{attribute 'no_explicit_call' := 'Do not call the body - Stick to OOP'}
FUNCTION_BLOCK FB_XTS_Mover EXTENDS FB_CH_Object IMPLEMENTS I_XTS_Mover, I_XTS_Mover_PLC
VAR	
	//Link to NC
	Axis : FB_XTS_Axis;

	{attribute 'hide'}
	bInitDone : BOOL;
	{attribute 'hide'}
	ipXtsSystem : I_XTS_System_Registration;
	{attribute 'hide'}
	ipUtilityMover : I_TcIoXtsXpuMover;
	{attribute 'hide'}
	ipProductData : I_XTS_ProductData; //later the required interface of the tool or product can be queried via query interface
	{attribute 'hide'}
	ipParentStation : I_XTS_Station; //This is the station in which the Mover is currently standing or moving.	
	{attribute 'hide'}
	ipNextMover : I_XTS_Mover;
	{attribute 'hide'}
	sTargedStation : STRING;
	{attribute 'hide'}
	fLastCmdTargedPosition : LREAL; //the last commanded target position [mm]
	{attribute 'hide'}
	fLastCmdTargedVelocity : LREAL; //the last commanded target speed
	{attribute 'hide'}	
	fLastCmdTargedGap 	: LREAL; //the last commanded target gap
	{attribute 'hide'}
	bInGroup : BOOL;	
	{attribute 'hide'}	
	lrTrackLentgh 			: LREAL; //[mm]  Modulo
	{attribute 'hide'}
	fbFeedback 					: CHALET_BaseComponents.FB_CH_Feedback(ipSourceInfo := fbSourceInfo);;
	
END_VAR
VAR PERSISTENT
	fDrivenDistance : LREAL;
END_VAR

{attribute 'monitoring':='call'}
PROPERTY Coupled : BOOL
GET
Coupled := THIS^.Axis.Coupled;
END_GET
END_PROPERTY

{attribute 'OPC.UA.DA.Property' := '1'}
{attribute 'monitoring':='call'}
PROPERTY DefaultAcceleration : LREAL
GET
DefaultAcceleration := THIS^.Axis.DefaultAcceleration;
END_GET
SET
THIS^.Axis.DefaultAcceleration := DefaultAcceleration;
END_SET
END_PROPERTY

{attribute 'OPC.UA.DA.Property' := '1'}
{attribute 'monitoring':='call'}
PROPERTY DefaultDeceleration : LREAL
GET
DefaultDeceleration := THIS^.Axis.DefaultDeceleration;
END_GET
SET
THIS^.Axis.DefaultDeceleration := DefaultDeceleration;
END_SET
END_PROPERTY

{attribute 'OPC.UA.DA.Property' := '1'}
{attribute 'monitoring':='call'}
PROPERTY DefaultJerk : LREAL
GET
DefaultJerk := THIS^.Axis.DefaultJerk;
END_GET
SET
THIS^.Axis.DefaultJerk := DefaultJerk;
END_SET
END_PROPERTY

METHOD Disable : HRESULT
Axis.PowerOff();


//Show as feedback the state of the includet axis
fbFeedback.ActiveCommand := Axis.Feedback.ActiveCommand;
fbFeedback.LastCommandAccepted := Axis.Feedback.LastCommandAccepted;
fbFeedback.HR := Axis.Feedback.hr;


IF Axis.Feedback.LastCommandAccepted THEN
	Disable := S_OK;
ELSE  
	Disable := E_FAIL;;	
END_IF
END_METHOD

{attribute 'monitoring':='call'}
PROPERTY DrivenDistance : LREAL
GET
DrivenDistance := fDrivenDistance;
END_GET
END_PROPERTY

METHOD Enable : HRESULT
Axis.PowerOn();


//Show as feedback the state of the includet axis
fbFeedback.ActiveCommand := Axis.Feedback.ActiveCommand;
fbFeedback.LastCommandAccepted := Axis.Feedback.LastCommandAccepted;
fbFeedback.HR := Axis.Feedback.hr;


IF Axis.Feedback.LastCommandAccepted THEN
	Enable := S_OK;
ELSE  
	Enable := E_FAIL;;	
END_IF
END_METHOD

METHOD FB_init : BOOL
VAR_INPUT
	bInitRetains : BOOL; // if TRUE, the retain variables are initialized (warm start / cold start)
	bInCopyCode : BOOL;  // if TRUE, the instance afterwards gets moved into the copy code (online change)
	
	ipXtsSystem : I_XTS_System_Registration; //Interface to XTS system object
END_VAR
VAR_INST
	{attribute 'hide'}
	bFBInitCalledOnce : BOOL; //Do the following code once during start up and not during onlinechange
END_VAR
//Do the following code once during start up and not during onlinechange
IF NOT bFBInitCalledOnce THEN 
	

	//Regristrate object in System
	IF ipXtsSystem <> 0 THEN
		ipXtsSystem.RegisterMover(THIS^);
		THIS^.ipXtsSystem := ipXtsSystem;
	END_IF


	
END_IF

bFBInitCalledOnce := TRUE;
END_METHOD

{attribute 'monitoring':='call'}
PROPERTY Feedback : I_CH_Feedback
GET
Feedback := THIS^.fbFeedback;
END_GET
END_PROPERTY

(*The _ PLC interface provides the user with a simplified interface for commanding between the stations. Sometimes, however, this is not enough. 
Either you get the corresponding interface with the __Queryinterface or you can get full access with this property.*)
PROPERTY FullAccess : I_XTS_Mover
GET
FullAccess := (THIS^);
END_GET
END_PROPERTY

PROPERTY getAxisRef : REFERENCE TO Tc2_MC2.AXIS_REF
GET
getAxisRef REF= THIS^.Axis.getAxisRef;
END_GET
END_PROPERTY

METHOD HaltCA : HRESULT
VAR_INPUT
END_VAR
Axis.HaltCA(
	fDeceleration:= 0, //use default
	fJerk:= 0, //use default
	fGap:= fLastCmdTargedGap);
	

//Show as feedback the state of the includet axis
fbFeedback.ActiveCommand := Axis.Feedback.ActiveCommand;
fbFeedback.LastCommandAccepted := Axis.Feedback.LastCommandAccepted;
fbFeedback.HR := Axis.Feedback.hr;


IF Axis.Feedback.LastCommandAccepted THEN
	HaltCA := S_OK;
ELSE  
	HaltCA := E_FAIL;;	
END_IF
END_METHOD

PROPERTY IdentInGroup : IDENT_IN_GROUP_REF
GET
IdentInGroup := UDINT_TO_IDENTINGROUP(THIS^.Axis.getAxisRef.NcToPlc.AxisId);
END_GET
END_PROPERTY

METHOD Initialize : HRESULT
VAR

END_VAR
fbFeedback.hr := S_OK;	

IF NOT THIS^.bInitDone THEN
	fbFeedback.ActiveCommand := 'Init';
	
	//Get Tracklength from system
	THIS^.lrTrackLentgh := THIS^.ipXtsSystem.TrackLength;
	
	
	//Validate Settings
	IF (lrTrackLentgh <= 0) THEN
		fbFeedback.hr := GetMostSignificant(fbFeedback.hr, E_FAIL);		
	END_IF
	

	//If only one mover is in project, then interface stays 0.
	IF THIS^.ipXtsSystem.Movers.Size > 1 THEN
		THIS^.ipNextMover := THIS^.ipXtsSystem.getMoverInFront(THIS^);
		//Validate Settings
		IF (ipNextMover = 0) THEN
			fbFeedback.hr := GetMostSignificant(fbFeedback.hr, E_FAIL);	
		END_IF
	ELSE
		THIS^.ipNextMover := 0;
	END_IF
	
	// Get XTS Utility mover object
	IF ipXtsSystem.Environment <> 0 THEN
		ipUtilityMover := ipXtsSystem.Environment.UtilityEnvirement.GetMoverInterfaceByAxisId(THIS^.getAxisRef.NcToPlc.AxisId);
		//Validate 
		IF (ipUtilityMover = 0) THEN
			fbFeedback.hr := GetMostSignificant(fbFeedback.hr, E_FAIL);	
		END_IF
	END_IF
	
	
	//InitAxis
	fbFeedback.hr := GetMostSignificant(fbFeedback.hr, Axis.Initialize());	

	bInitDone := CheckOk(fbFeedback.hr);
END_IF

Initialize := fbFeedback.hr;
END_METHOD

{attribute 'monitoring':='call'}
PROPERTY LagDistance : LREAL
GET
LagDistance := THIS^.Axis.LagDistance;
END_GET
END_PROPERTY

{attribute 'monitoring':='call'}
PROPERTY LastCmdTargedGap : LREAL
GET
LastCmdTargedGap := fLastCmdTargedGap;
END_GET
END_PROPERTY

{attribute 'monitoring':='call'}
PROPERTY LastCmdTargedPosition : LREAL
GET
LastCmdTargedPosition := fLastCmdTargedPosition;
END_GET
END_PROPERTY

{attribute 'monitoring':='call'}
PROPERTY LastCmdTargedVelocity : LREAL
GET
LastCmdTargedVelocity := fLastCmdTargedVelocity;
END_GET
END_PROPERTY

METHOD MoveAbsCA : HRESULT
VAR_INPUT
	fPosition	: LREAL := MC_INVALID;
	fVelocity	: LREAL := MC_INVALID;
	fGap		: LREAL := MC_DEFAULT;
	eDirection	: Tc3_Mc3Definitions.MC_DIRECTION;
END_VAR
Axis.MoveAbsoluteCA(
	fPosition:= fPosition, 
	fVelocity:= fVelocity, 
	fGap:= fGap, 
	fAcceleration:= 0, //Use Axis default
	fDeceleration:= 0, //Use Axis default
	fJerk:= 0, 			//Use Axis default
	eDirection := eDirection,
	eBufferMode:= Tc3_Mc3Definitions.MC_BUFFER_MODE.mcAborting);

THIS^.fLastCmdTargedVelocity := fVelocity;
THIS^.fLastCmdTargedPosition := fPosition;
THIS^.fLastCmdTargedGap := fGap;


//Show as feedback the state of the includet axis
fbFeedback.ActiveCommand := Axis.Feedback.ActiveCommand;
fbFeedback.LastCommandAccepted := Axis.Feedback.LastCommandAccepted;
fbFeedback.HR := Axis.Feedback.hr;


IF Axis.Feedback.LastCommandAccepted THEN
	MoveAbsCA := S_OK;
ELSE  
	MoveAbsCA := E_FAIL;;	
END_IF
END_METHOD

{attribute 'monitoring':='call'}
PROPERTY MoverInGroup : BOOL
GET
MoverInGroup := bInGroup;
END_GET
SET
bInGroup := MoverInGroup;
END_SET
END_PROPERTY

{attribute 'monitoring':='call'}
PROPERTY Moving : BOOL
GET
Moving := THIS^.Axis.Moving;
END_GET
END_PROPERTY

{attribute 'monitoring':='call'}
PROPERTY NextMover : I_XTS_Mover
GET
NextMover := ipNextMover;
END_GET
END_PROPERTY

{attribute 'monitoring':='call'}
PROPERTY OID : OTCID
GET
OID := THIS^.Axis.OID;
END_GET
END_PROPERTY

{attribute 'monitoring':='call'}
PROPERTY ParentStation : I_XTS_Station
GET
ParentStation := ipParentStation;
END_GET
SET
ipParentStation := ParentStation;
END_SET
END_PROPERTY

{attribute 'monitoring':='call'}
PROPERTY PositionOnTrack : LREAL
GET
//Round to 3 digits. If Axis is not enabled, use act position
IF THIS^.Axis.getAxisRef.Status.Disabled THEN
	PositionOnTrack := TO_LREAL(TRUNC(THIS^.Axis.ActPosModulo*1000))/1000;
ELSE
	PositionOnTrack := TO_LREAL(TRUNC(THIS^.Axis.SetPosModulo*1000))/1000;	
END_IF
END_GET
END_PROPERTY

{attribute 'monitoring':='call'}
PROPERTY PUBLIC ProductData : I_XTS_ProductData
GET
ProductData := ipProductData;
END_GET
SET
// No change. Same interface is set again
IF ipProductData = ProductData THEN
	;//Noting
	
ELSE

	// If allready an interface is linked. Unlink
	IF ipProductData <> 0 THEN
		ipProductData.LinkToMover(0);
		ipProductData := 0;
	END_IF
	
	// Link and store new interface
	IF ProductData <> 0 THEN
		ProductData.LinkToMover(THIS^);
		ipProductData := ProductData;
	END_IF
END_IF
END_SET
END_PROPERTY

METHOD Reset : HRESULT
Axis.Reset();

//Show as feedback the state of the includet axis
fbFeedback.ActiveCommand := Axis.Feedback.ActiveCommand;
fbFeedback.LastCommandAccepted := Axis.Feedback.LastCommandAccepted;
fbFeedback.HR := Axis.Feedback.hr;


IF Axis.Feedback.LastCommandAccepted THEN
	Reset := S_OK;
ELSE  
	Reset := E_FAIL;;	
END_IF
END_METHOD

{attribute 'monitoring':='call'}
PROPERTY SetAcceleration : LREAL
GET
SetAcceleration := THIS^.Axis.SetAcceleration;
END_GET
END_PROPERTY

{attribute 'monitoring':='call'}
PROPERTY SetVelocity : LREAL
GET
SetVelocity := THIS^.Axis.SetVelocity;
END_GET
END_PROPERTY

{attribute 'monitoring':='call'}
PROPERTY TargedStation : STRING
GET
TargedStation := sTargedStation;
END_GET
SET
sTargedStation := TargedStation;
END_SET
END_PROPERTY

METHOD Update : HRESULT
VAR
	fDistanceThisCycle : LREAL;
END_VAR
VAR_INST
	fLastMoverPosition : LREAL;
END_VAR
// Total distance traveled by the mover
IF Axis.Moving THEN
	fDistanceThisCycle := ABS(Axis.SetPosModulo-fLastMoverPosition);
	IF fDistanceThisCycle > (THIS^.lrTrackLentgh*0.5) THEN
		fDistanceThisCycle := THIS^.lrTrackLentgh-fDistanceThisCycle;
	END_IF
	fDrivenDistance := fDrivenDistance + fDistanceThisCycle;
END_IF

fLastMoverPosition := Axis.SetPosModulo;

Axis.Update();

//Show as feedback the state of the includet axis
fbFeedback.ActiveCommand := Axis.Feedback.ActiveCommand;
fbFeedback.HR := Axis.Feedback.hr;
END_METHOD

{attribute 'monitoring':='call'}
PROPERTY UtilityMover : I_TcIoXtsXpuMover
GET
UtilityMover := ipUtilityMover;
END_GET
END_PROPERTY

END_FUNCTION_BLOCK

(* stored: Version 1.1.0.1, ProductVersion 3.1.4024.12
   POU FB_XTS_Mover: Id {3ed790a4-6e64-4b54-8db7-341624f96fe6}, SpecialFunc None
   Folder Command: Id {ca288374-806c-40ea-bc74-0ab5bbcbeeac}
   Folder Dynamics: Id {b9fcfb38-b272-4ca4-b13a-341f5f54d90d}
   Folder Status: Id {36fbca5a-40fa-4fee-a207-226360d4b0d4}
   Property Coupled: Id {627291ab-402b-4929-a093-0ff8fc3ea751}
   Get Get: Id {f28a9d3d-b665-4255-8ee8-a1611de68e13}
   Property DefaultAcceleration: Id {18610012-8a94-4ab6-bb6e-6d4fcc935be7}
   Get Get: Id {30c1feb4-1bec-4b32-8312-941a2f3f97e6}
   Set Set: Id {73641ac0-c47d-4373-aafd-c8aa42e11a4f}
   Property DefaultDeceleration: Id {a4e01ee3-7720-44ba-aa6b-afa8d7117cca}
   Get Get: Id {ff90a48b-809c-4768-9581-05a95fc76f54}
   Set Set: Id {ecb6ccf7-e313-4889-af0f-b2b90db416f6}
   Property DefaultJerk: Id {d2dd93df-7379-493e-a0e2-335666e5944c}
   Get Get: Id {9bcab0a6-60f8-42f0-9374-f84d6b198092}
   Set Set: Id {5eea3280-3211-4781-b593-3f1678c35bbf}
   Method Disable: Id {fabc84ce-66bc-42ad-9f05-26b65256e1b0}
   Property DrivenDistance: Id {b520ba11-eae3-4194-b965-36b18e5c7ced}
   Get Get: Id {713472d5-7bea-4713-b937-1508a3c15ef1}
   Method Enable: Id {c5208f99-fcd6-4588-ba54-a943e08cbd2d}
   Method FB_init: Id {26d010fc-cadf-4788-a716-5e39c9198509}
   Property Feedback: Id {78e76366-75b3-4e4d-b82e-9b66faf8cccb}
   Get Get: Id {53c4eaab-cafe-47f9-880a-ceebaeabf33e}
   Property FullAccess: Id {0cd8020e-3c30-4c65-a148-8455972ce3b7}
   Get Get: Id {dc1cc900-5ae5-4ac7-b5fd-19291576e9ec}
   Property getAxisRef: Id {e9338665-6fdb-4597-a49b-106d166a108b}
   Get Get: Id {380384b0-402e-4f2b-b606-a794dede7c6a}
   Method HaltCA: Id {b3b73891-2843-460d-b720-beb958a16aee}
   Property IdentInGroup: Id {16fd8e53-436d-4269-afa6-4835331c3eb4}
   Get Get: Id {66d1a06a-a12e-497f-9136-eb6174f741d0}
   Method Initialize: Id {23d9f9f9-f9dc-4f21-803f-f56ae726981f}
   Property LagDistance: Id {fa2169ed-cf4a-4db4-abdd-b47bb25a427a}
   Get Get: Id {481cd61e-87a5-4a23-802c-06c901cb6898}
   Property LastCmdTargedGap: Id {c603e157-0a0b-4fe1-aa25-9803f19d5a3b}
   Get Get: Id {86180dea-72a2-44e5-98be-24c2f95a6f1f}
   Property LastCmdTargedPosition: Id {3958310d-6370-4bc5-9821-b9fcf79326a2}
   Get Get: Id {0cc8ea36-ff74-4575-81b6-5407cf19e616}
   Property LastCmdTargedVelocity: Id {1b8ff9df-ff49-4e9c-9925-a9f950566659}
   Get Get: Id {6d914134-e0b8-4a08-ba17-5ff68a157872}
   Method MoveAbsCA: Id {e608c39d-112a-4026-931d-1e2e9427af10}
   Property MoverInGroup: Id {1456bf31-7e86-484b-b915-73afc447ac11}
   Get Get: Id {0f057045-f770-4314-b040-34f6e64174be}
   Set Set: Id {3c0acef1-3a7f-4a39-8b35-c7b1fc94d122}
   Property Moving: Id {7f684ea5-18fb-4113-9f2e-3e6e6516eb36}
   Get Get: Id {b6a0da70-c417-4d3b-ba79-4206b4ba4722}
   Property NextMover: Id {cfe98c85-e400-447d-84c6-6a0d712a3ba3}
   Get Get: Id {d18cdb15-51fd-4bb2-8b90-9e642aa239cc}
   Property OID: Id {fff58861-514a-439b-92c4-eaf63536f340}
   Get Get: Id {a17ad2ef-7302-4629-9cd9-0e4f954bfad3}
   Property ParentStation: Id {6cca7d79-22b7-4800-bcd7-e5da152983ec}
   Get Get: Id {dfe80be0-f7f8-476a-b158-3b9e081323d5}
   Set Set: Id {59bbc721-c9b4-4d89-b456-547c6ecc3201}
   Property PositionOnTrack: Id {3c69251b-801e-4c6a-b612-567ec3e5bf9f}
   Get Get: Id {e39d0e2b-c78c-4fa5-acc7-b84c6e63f69f}
   Property ProductData: Id {389f0e05-56fd-43ad-a266-706c31820384}
   Get Get: Id {019d049e-dcda-4c9d-91ee-9f7c613d9e2f}
   Set Set: Id {3c645bf0-f6f5-45e0-a21c-f1f84867eff3}
   Method Reset: Id {105a8a39-edcf-452e-8280-230926f87f92}
   Property SetAcceleration: Id {8a067508-9273-45b2-a870-3d2124b777fa}
   Get Get: Id {2198d9cd-6a99-433b-877e-25b3061464bd}
   Property SetVelocity: Id {61dc005e-7627-4d18-968d-6cc1c0e072c5}
   Get Get: Id {bf4b231b-d926-4778-8d14-891d71bd7807}
   Property TargedStation: Id {47a0a370-02c4-4535-9177-11a7259d5869}
   Get Get: Id {a49a56c6-50fe-424b-a33a-79d1d1912a0d}
   Set Set: Id {19ab049a-80fc-44a6-a298-d92eea4f119a}
   Method Update: Id {c49f710e-dc5c-4925-a604-489fc7b469ad}
   Property UtilityMover: Id {98bbafb7-19de-441a-bce6-57eeb214e8c0}
   Get Get: Id {d02bd165-9926-40b8-af38-1d5af2ae164e} *)
